{attribute 'qualified_only'}
// ***********************************************************************************
//
// Müller-steinag Gruppe, Kandergrien Einigen, CH-3646 Bern
// ETH Zurich, Building HIF E26, Laura-Hezner-Weg 7, CH-8093 Zürich
// 
// ***********************************************************************************
// 
// PROJECT     :  A061 Digital Casting System 
// FUNCTION    :  Profinet Variable Convertor
// AUTHOR      :  Weiting Chen
// EMAIL       :  chenw@usi.ch
// Copyright   :  USI Mendrisio; ETH Zürich; Müller-steinag Gruppe (CH) 2023
// Contributor :  Fabio Scotto / Philippe Fleischmann 
//
// ***********************************************************************************

VAR_GLOBAL
//
//File description 
//GVL(GVL : Global variables)
//GVL_IO(GVL_IO : IO)
//GVL_PN(GVL_PN : Profinet Array)
//GVL_RED(GVL_research : variables for control via laptop)
//GVL_ROB(GVL_research : variables for control via Robot)

//
//Data Type Prefix
//ib = Input Bool   / ob = Output Bool
//if = Input float  / of = Output float (REAL, LREAL)
//in = Input numeric/ on = Output numeric 
//(INT, SINT, USINT, UNIT, DINT, UDINT, BYTE, WORD, DWORD, LWORD, XINT, UXINT, XWORD) 
//t = Time (TON)
//s = String

//
//Naming Shortcuts
//CC1 = Concrete Controller 
//AP1 = Admixture pump, High dosage ViscoTech Pump (Xseed or Accelerator)
//CP1 = Concrete Pump
//SP1 = Admixture pump, Low dosage ViscoTech Pump  (Xseed or Accelerator or Superplasticizer)

//PP1 = Peristaltic Pump
//MI1 = Mixer
//T1  = Tool 1
//CA1 = Camera 1
//RED = Research Data
//PN = Profinet with Roboter

END_VAR

(* stored: Version 1.1.0.1, ProductVersion 3.1.4024.11
   GVL ReadMe: Id {6354b487-1c67-4bd0-bfdf-078ef0b6da95} *)
